RoboDK station: ) — копия — копия.rdk

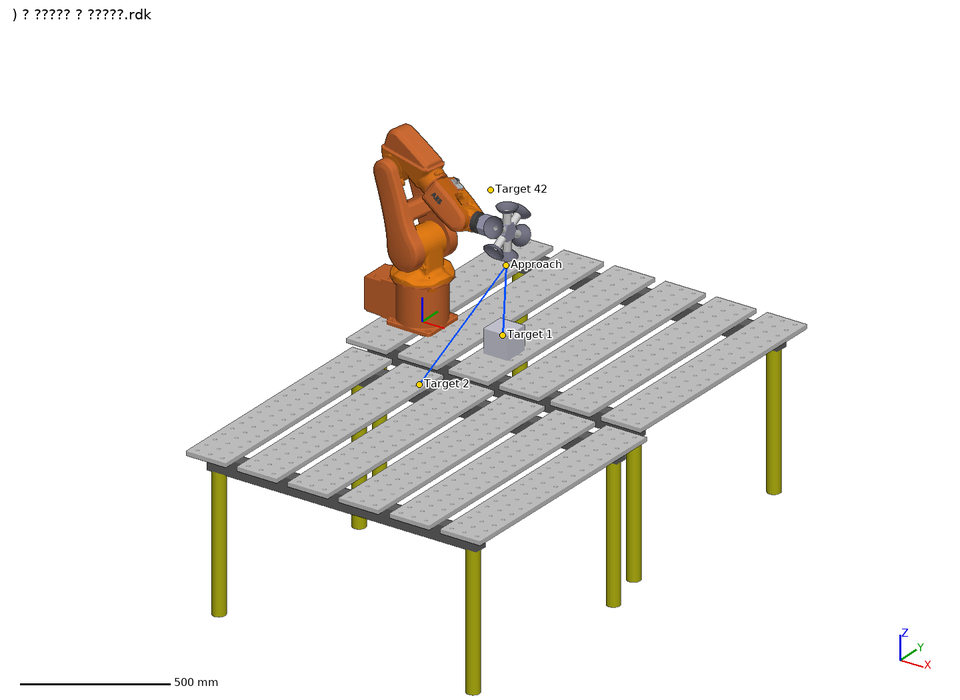
[picture v0: the station drawn from its stored meshes, robots at their saved joint values, targets as dots, program paths as lines]
Station ). Poses are relative to the parent item; angles as X-Y-Z fixed-axis rotations.
  - frame ABB IRB 120-3/0.6 Base at (60.92, -16.78, 0) mm
    - robot ABB IRB 120-3/0.6: 6 axes, payload 3 kg, reach 580 mm, repeatability 0.01 mm, weight 25 kg
        modified DH rows (alpha deg, a mm, theta deg, d mm): 0, 0, 0, 290; -90, 0, -90, 0; 0, 270, 0, 0; -90, 70, 0, 302; 90, 0, 0, 0; -90, 0, 180, 72
        joint limits [-165, -110, -90, -160, -120, -400] to [165, 110, 70, 160, 120, 400]; home [0, 0, 0, 0, 0, 0]; saved at [-9.453, -21.494, 51.842, -18.239, -31.652, 15.67]
      - tool Tool, TCP at (125, -3.56, 100) mm, rotated rx 0 ry 90 rz 0 deg, size 184.7 x 197.7 x 137.7 mm
      - tool TCP 1, TCP at (73.87, -0.56, 98.27) mm
    - target Target 2 (Cartesian target) at (338.43, -501.58, 60.32) mm, rotated rx -180 ry 0 rz -180 deg; joints [-71.521, 76.956, -31.613, -76.628, -77.128, 43.142] of ABB IRB 120-3/0.6
    - target Target 1 (Cartesian target) at (352.26, -36.32, 62.02) mm, rotated rx 180 ry 0 rz 180 deg; joints [-10.3, 39.985, 61.269, -10.497, -101.07, -2.038] of ABB IRB 120-3/0.6
    - frame Frame pick and place at (0, 0, 0) mm
      - object Table at (462.97, 233.54, 0) mm, size 1193.8 x 965.2 x 609.6 mm, geometry from welding_table.sld
    - target Approach (Cartesian target) at (366.38, -35.93, 324.04) mm, rotated rx 180 ry 0 rz 180 deg; joints [-9.453, -21.494, 51.842, -18.239, -31.652, 15.67] of ABB IRB 120-3/0.6
    - frame Frame 2 at (0, 0, 0) mm
      - object Table at (516.25, -773.06, 0) mm, size 1193.8 x 965.2 x 609.6 mm, geometry from welding_table.sld
    - target Target 42 (Cartesian target) at (309.94, -45.15, 590.28) mm, rotated rx 180 ry 0 rz -180 deg; joints [-16.776, -23.909, 1.816, -141.288, -27.484, 144.585] of ABB IRB 120-3/0.6
  - program pick and place (14 instructions, listed below)
  - program Replace objects (1 instructions, listed below)
  - object box at (415.51, -49.57, 42.59) mm, size 100 x 100 x 100 mm, geometry from box.sld
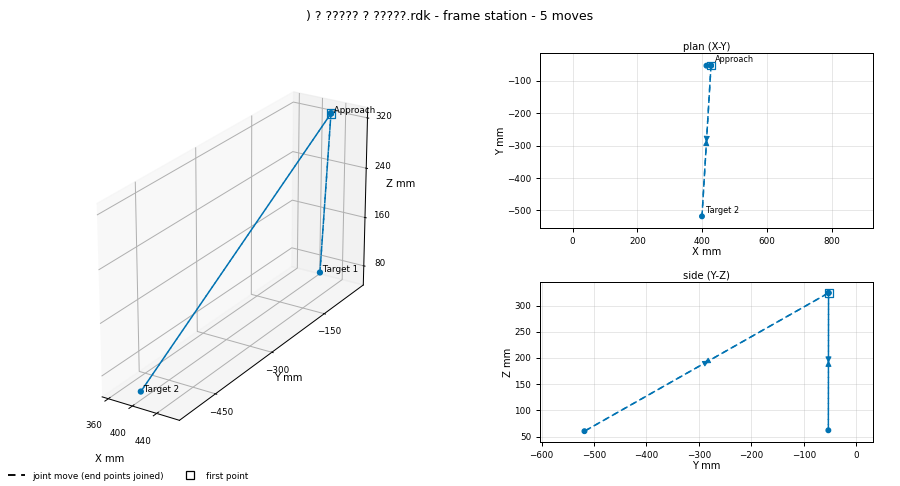
[picture p0: tool path of ) — копия — копия.rdk in frame station, 5 of 5 moves have a stored position in this frame; points joined in program order, loops and branches not executed]

--- program pick and place (robot ABB IRB 120-3/0.6) ---
  Set speed (50.0 mm/s)
  Set Ref.: Frame pick and place
  Set Tool: Tool
  MoveJ (Approach)
  MoveJ (Target 1)
  Attach to Tool
  Call AirValve_On
  MoveJ (Approach)
  Change Frame -> Frame 2
  MoveJ (Target 2)
  Detach from Tool
  Call AirValve_Off
  MoveJ (Approach)
  Call Replace objects

--- program Replace objects (robot ABB IRB 120-3/0.6) ---
  Replace objects
